TYPE ST_HMIComponentAPI :
STRUCT 
	Done : BOOL;
	Busy : BOOL;
	Error : BOOL;
	ErrorID : BOOL;
	Ready : BOOL;
	Enabled: BOOL;
	Homed: BOOL;
	Moving : BOOL;
END_STRUCT
END_TYPE

(* stored: Version 1.1.0.1
   DUT ST_HMIComponentAPI: Id {de9cb45b-e895-47f7-93d7-0e4ccd710743} *)
